// TIA Portal V16 export
// export: Created 2021-05-25T16:14:40.2760782Z, ExportSetting WithDefaults, DisplayName Totally Integrated Automation Portal, DisplayVersion V16, DisplayName TIA Portal Version Control Interface, DisplayVersion V16, DisplayName TIA Portal Openness, DisplayVersion V16, DisplayName STEP 7 Professional, DisplayVersion V16, DisplayName STEP 7 Safety, DisplayVersion V16, DisplayName WinCC Unified SCADA Engineering System, DisplayVersion V16
DATA_BLOCK "dbDigitalValves"   // DB32
{ S7_Optimized_Access := 'FALSE'; DB_Accessible_From_OPC_UA := 'FALSE' }
VERSION : 0.1
// stored: AutoNumber false, DBAccessibleFromOPCUA false, IsOnlyStoredInLoadMemory false, IsWriteProtectedInAS false
   VAR
      Y17_RotCilipozDesno : "udtDigitalValve";   // Crane control not selected lamps (Q0.0)
      Y18_RotCilipozLevo : "udtDigitalValve";
      Y2_VijaDesZad_Dvig : "udtDigitalValve";
      Y3_VijaDesSpr_Dvig : "udtDigitalValve";
      Y4_VijaLevZad_Dvig : "udtDigitalValve";
      Y5_VijaLevSpr_Dvig : "udtDigitalValve";
      Y6_DrcaLocev_Des : "udtDigitalValve";
      Y7_DrcaLocev_Lev : "udtDigitalValve";
      Y8_VijaLocev_Des : "udtDigitalValve";
      Y9_VijaStop_DesZad : "udtDigitalValve";
      Y10_Centri_DesZad : "udtDigitalValve";
      Y11_Centri_DesSpr : "udtDigitalValve";
      Y12_VijaLocev_Lev : "udtDigitalValve";
      Y13_VijaStop_LevZad : "udtDigitalValve";
      Y14_Centri_LevZad : "udtDigitalValve";
      Y15_Centri_LevSpr : "udtDigitalValve";
      Y16_VpenjanjeDna : "udtDigitalValve";
      SEMAFOR_ZELENA : "udtDigitalValve";
      SEMAFOR_RUMENA : "udtDigitalValve";
      SEMAFOR_RDECA : "udtDigitalValve";
   END_VAR
BEGIN
END_DATA_BLOCK
